FUNCTION TryConvert_BYTE_TO_UDINT : BOOL
VAR_INPUT
	in : BYTE;
	out : REFERENCE TO UDINT;
END_VAR

out := BYTE_TO_UDINT(in);
TryConvert_BYTE_TO_UDINT := TRUE;

END_FUNCTION

(* stored: Version 1.1.0.1, ProductVersion 3.1.4024.12
   POU TryConvert_BYTE_TO_UDINT: Id {b5357d5c-55e3-43ab-865f-a4f06a425048}, SpecialFunc None *)
